(* CODESYS project Tc3_Element.library
   Description: State Model with Observer and Events
   Author: Peter Zerlauth
   Company: Zerlauth
   Version: 0.0.0.1
   Title: Tc3_Element
   DefaultNamespace: Tc3_Element
   Placeholder: Tc3_Element

Project tree, tasks and I/O mapping:
  libraries: Tc2_Standard, * (Beckhoff Automation GmbH); Tc2_System, * (Beckhoff Automation GmbH); Tc2_Utilities, * (Beckhoff Automation GmbH); Tc3_Module, 3.4.5.0 (Beckhoff Automation GmbH)
  Element/
    Event/
      Observable/
        function block FB_Observable [ST]: FB_exit, M_Attach, M_Clear, M_Detach, M_Find, M_Index, M_Notify, P_Length
        interface I_Observable: M_Attach, M_Detach, P_Length
        interface I_Observer: M_Notify
      data type E_Event
      data type E_EventType
      function block FB_Event [ST]: FB_init, M_Abort, M_AddBOOL, M_AddINT, M_AddREAL, M_AddSTRING, M_AddTIME, M_Arguments, M_Build, M_Debug, M_Error, M_Info, M_Log, M_Warning, P_Logger, P_Observer
      interface I_Event: M_Abort, M_AddBOOL, M_AddINT, M_AddREAL, M_AddSTRING, M_AddTIME, M_Debug, M_Error, M_Info, M_Warning, P_Logger, P_Observer
      data type ST_Event
      data type ST_EventFlags
    Reflection/
      function block FB_Reflection [ST]: M_GetInstance, P_Class, P_Comment, P_ID, P_Instance, P_Timestamp
      interface I_Reflection : P_Class, P_Comment, P_ID, P_Instance, P_Timestamp
    Sequence/
      data type E_Sequence
      function block FB_Sequence [ST]: FB_init, M_Await, M_Reset, M_Restore, M_Set, P_Number, P_Timeout
      interface I_Sequence: M_Await, M_Reset, M_Set, P_Number, P_Timeout
      data type ST_Sequence
      data type ST_SequenceOptions
    data type E_Request
    data type E_State
    function block FB_Element [ST]: M_Aborted, M_Aborting, M_Completed, M_Completing, M_Execute, M_Held, M_Holding, M_Idle, M_Paused, M_Pausing, M_Resetting, M_Resuming, M_Starting, M_Stopped, M_Stopping, M_Unholding, M_OnState, M_Request, P_Event, P_Reflection, P_Sequence, P_State
    interface I_Element: M_Request, P_Event, P_Reflection, P_State
  Level/
    function block FB_Level [ST]: M_Aborting, M_Attach, M_Completing, M_Detach, M_Holding, M_Pausing, M_Resetting, M_Resuming, M_Starting, M_Stopping, M_Unholding, P_List
  List/
    function block FB_ListElement [ST]: FB_exit, M_Add, M_Clear, M_Find, M_Index, M_Remove, P_Length
    function block FB_ListObject [ST]: FB_exit, M_Add, M_Clear, M_Find, M_Index, M_Remove, P_Length
    function block FB_ListString [ST]: FB_exit, M_Add, M_Clear, M_Find, M_Index, M_Remove, P_Length
    interface I_ListBase: M_Clear, P_Length
    interface I_ListElement: M_Add, M_Find, M_Index, M_Remove
    interface I_ListObject: M_Add, M_Find, M_Index, M_Remove
    interface I_ListString: M_Add, M_Find, M_Index, M_Remove
  Logger/
    function block FB_FileLogger [ST]: M_Delete, M_Find, M_Log, M_Reset
    function block FB_Logger [ST]: M_Delete, M_Find, M_Log, M_Reset
    function block FB_LoggingProvider [ST]: FB_exit, M_Add, M_Clear, M_Find, M_Index, M_Log, M_Remove, M_Reset, P_Length
    interface I_Logger: M_Log, M_Reset
  Module/
    data type E_Mode
    function block FB_Module [ST]: M_Aborting, M_Completing, M_Holding, M_Idle, M_Mode, M_OnMode, M_Resetting, M_Starting, M_Stopping, M_Unholding, P_Mode
    interface I_Module: M_Mode, P_Mode
  Object/
    function block FB_Object [ST]
    interface I_Object
  Utils/
    File/
      function block FB_File [ST]: M_Append, M_AppendLine, M_Close, M_Create, M_Delete, M_Load, M_Open, M_Read, M_Write, P_Error, P_Open
      interface I_File: M_Append, M_AppendLine, M_Close, M_Create, M_Delete, M_Load, M_Open, M_Read, M_Write, P_Error, P_Open
    function block FB_Debounce [ST]: P_Value
  Version/
    global variables Global_Version
*)

// Element/Event/E_Event
{attribute 'qualified_only'}
{attribute 'strict'}
{attribute 'to_string'}
TYPE E_Event :
(
	Verbose			:= 0,
	Debug			:= 1,
	Information		:= 2,
	Warning			:= 3,
	Error			:= 4
);
END_TYPE

// Element/Event/E_EventType
{attribute 'qualified_only'}
{attribute 'strict'}
{attribute 'to_string'}
TYPE E_EventType :
(
	Information		:= 1,
	Warning			:= 2,
	Stop			:= 3,
	Abort			:= 4
);
END_TYPE

// Element/Event/ST_Event
{attribute 'analysis' := '-33'}
TYPE ST_Event :
	STRUCT
		iSource:		I_Element;
		eEventType:		E_Event;
		tTimestamp:   	DT;
		nID:			ULINT;
		sInstance:		STRING(255);
		sClass:			STRING(255);
		sMessage:		STRING(255);
		sDefault:		STRING(255);
		sArguments:		STRING(255);
   		{attribute 'hide'} 
		stFlags:		ST_EventFlags;
	END_STRUCT
END_TYPE

// Element/Event/ST_EventFlags
{attribute 'analysis' := '-33'}
TYPE ST_EventFlags :
STRUCT
	bActive:		BIT;
	bRemove:		BIT;
END_STRUCT
END_TYPE

// Element/Sequence/E_Sequence
{attribute 'qualified_only'}
{attribute 'strict'}
{attribute 'to_string'}

TYPE E_Sequence :
(
	Undefined		:= -32767,
	Start			:= 0,
	Done			:= 32767
)INT;
END_TYPE

// Element/Sequence/ST_Sequence
TYPE ST_Sequence :
STRUCT
	sMessage:				STRING(255);
	nNumber:				INT;
END_STRUCT
END_TYPE

// Element/Sequence/ST_SequenceOptions
TYPE ST_SequenceOptions :
STRUCT
	bSaveOnStopping:		BOOL;
END_STRUCT
END_TYPE

// Element/E_Request
{attribute 'qualified_only'}
{attribute 'strict'}
{attribute 'to_string'}

TYPE E_Request :
(
	{attribute 'hide'}
    Undefined   := 0,
	{attribute 'analysis' := '-27'}
	Reset       := 1,
	{attribute 'analysis' := '-27'}
    Start       := 2,
	{attribute 'analysis' := '-27'}
	Pause		:= 4,
	{attribute 'analysis' := '-27'}
	Hold		:= 5,
	{attribute 'analysis' := '-27'}
	Complete	:= 6,
	{attribute 'analysis' := '-27'}
	Stop		:= 7,
	{attribute 'analysis' := '-27'}
	Abort		:= 8
);
END_TYPE

// Element/E_State
{attribute 'qualified_only'}
{attribute 'strict'}
{attribute 'to_string'}
TYPE E_State :
(
    Resetting       := -1,
   	Idle            := 0,
    Starting        := 1,
    Execute         := 2,
	Pausing			:= 3,
	Paused			:= 4,
	Resuming		:= 5,
	Holding			:= 6,
	Held			:= 7,
	Unholding		:= 8,
    Completing      := 9,
    Completed       := 10,
    Stopping        := 11,
    Stopped         := 12,
    Aborting        := 13,
    Aborted         := 14

)INT;
END_TYPE

// Module/E_Mode
{attribute 'qualified_only'}
{attribute 'strict'}
{attribute 'to_string'}
TYPE E_Mode :
(
	{attribute 'hide'}
    Undefined   := 0,
	Automatic   := 1,
    Semiauto    := 2,
	Manual		:= 3
);
END_TYPE

// Version/Global_Version
{attribute 'TcGenerated'}
{attribute 'no-analysis'}
{attribute 'linkalways'}
// This function has been automatically generated from the project information.
VAR_GLOBAL CONSTANT
	{attribute 'const_non_replaced'}
	stLibVersion_Tc3_Element : ST_LibVersion := (iMajor := 0, iMinor := 0, iBuild := 0, iRevision := 1, nFlags := 0, sVersion := '0.0.0.1');
END_VAR

// Element/Event/Observable/FB_Observable
FUNCTION_BLOCK PUBLIC FB_Observable IMPLEMENTS I_Observable
VAR_INPUT
	iParent:		I_Element;	
END_VAR
VAR
	bObserver:		BOOL;
	pList: 			POINTER TO I_Element;
    {attribute 'hide'}
	nLength:		DINT;
	{IF (defined (release))}
    	{attribute 'hide'}
	{END_IF}
	aList:			POINTER TO POINTER TO ARRAY [0..100] OF I_Element:=ADR(pList);
END_VAR

// https://peterzerlauth.com/
bObserver:= TRUE;

METHOD FB_exit : BOOL
VAR_INPUT
	bInCopyCode : BOOL; // if TRUE, the exit method is called for exiting an instance that is copied afterwards (online change).
END_VAR
M_Clear();
END_METHOD

METHOD M_Attach : BOOL
VAR_INPUT
	iObject: 	I_Element;
END_VAR
VAR
	pOldList: 	POINTER TO I_Element;
END_VAR
IF iObject <> 0 THEN
	// First Item
	IF pList = 0 THEN
		nLength:= nLength + 1;
		pList:= __NEW(POINTER TO I_Element,DINT_TO_UDINT(nLength));
	ELSE
		// Item already in List
		IF M_Find(iObject) = -1 THEN
			// backup 
			pOldList:= pList;
			// new Length
			nLength:= nLength + 1;
			// new pointer
			pList:= __NEW(POINTER TO I_Element,DINT_TO_UDINT(nLength));
			// restore
			Memcpy(pList,pOldList, SIZEOF(POINTER TO I_Element)*DINT_TO_UDINT(nLength -1));
			// delete old
			__DELETE(pOldList);
		ELSE
			M_Attach:= FALSE;	
			RETURN;
		END_IF
	END_IF
	IF pList = 0 THEN
		RETURN;
	END_IF
	// add new Object
	pList[nLength-1]:= iObject;
	M_Attach:= TRUE;
ELSE
	M_Attach:= FALSE;	
END_IF
END_METHOD

METHOD M_Clear
IF pList <> 0 THEN
	nLength:= 0;
	__DELETE(pList);
END_IF
END_METHOD

METHOD M_Detach : BOOL
VAR_INPUT
	iObject: 	I_Element;
END_VAR
VAR
	pOldList:			POINTER TO I_Element;
	nPosition: 			DINT;
END_VAR
IF iObject <> 0 THEN
	// First Item
	IF nLength >= 0 THEN
		// Item already in List
		nPosition:= M_Find(iObject);
		IF nPosition <> -1 THEN
			// backup 
			pOldList:= pList;
			// new Length
			nLength:= nLength -1;
			// new pointer
			pList:= __NEW(POINTER TO I_Element,DINT_TO_UDINT(nLength));
			// restore lower part
			Memcpy(pList,pOldList, SIZEOF(POINTER TO I_Element) * DINT_TO_UDINT(nPosition));
			//pList[nPosition]:= iObject;
			Memcpy(pList + (SIZEOF(POINTER TO I_Element)*nPosition),pOldList + (SIZEOF(POINTER TO I_Element)*(nPosition + 1)), SIZEOF(POINTER TO I_Element) * DINT_TO_UDINT(nLength - nPosition));
			// delete old
			__DELETE(pOldList);
		ELSE
			M_Detach:= FALSE;	
			RETURN;
		END_IF
	ELSE
		M_Detach:= FALSE;	
		RETURN;
	END_IF
	M_Detach:= TRUE;
ELSE
	M_Detach:= FALSE;	
END_IF
END_METHOD

METHOD M_Find : DINT
VAR_INPUT
	iObject: 	I_Element;
END_VAR
VAR
	nIndex: 	UINT;
END_VAR
// Object already in List
M_Find := -1;
WHILE nIndex < nLength DO
    IF (pList[nIndex] = iObject) THEN
        M_Find := nIndex;
        RETURN;
    END_IF
	nIndex := nIndex + 1;
END_WHILE
END_METHOD

METHOD M_Index : I_Observer
VAR_INPUT
	nIndex: 	DINT;
END_VAR
IF nIndex <= nLength THEN
	M_Index:= pList[nIndex].P_Event.P_Observer;
END_IF
END_METHOD

METHOD M_Notify
VAR_INPUT
	iSender:		I_Element;
END_VAR

VAR
	nIndex: 		DINT;
END_VAR
iParent.M_Request(E_Request.Abort);
IF bObserver THEN
	bObserver:= FALSE;
	WHILE nIndex < nLength DO
		pList[nIndex].P_Event.P_Observer.M_Notify(iSender);	
		nIndex:= nIndex + 1; 
	END_WHILE
	
END_IF
END_METHOD

{attribute 'OPC.UA.DA.Property' := '1'}
{attribute 'monitoring' := 'call'}
PROPERTY P_Length : DINT
GET
P_Length:= nLength;
END_GET
END_PROPERTY

END_FUNCTION_BLOCK

// Element/Event/Observable/I_Observable
INTERFACE I_Observable EXTENDS I_Observer

METHOD PUBLIC M_Attach : BOOL
VAR_INPUT
	iObject: 	I_Element;
END_VAR
END_METHOD

METHOD PUBLIC M_Detach : BOOL
VAR_INPUT
	iObject: 	I_Element;
END_VAR
END_METHOD

{attribute 'OPC.UA.DA.Property' := '1'}
{attribute 'monitoring' := 'call'}
PROPERTY P_Length : DINT
GET
END_GET
END_PROPERTY

END_INTERFACE

// Element/Event/Observable/I_Observer
INTERFACE I_Observer EXTENDS I_Object

METHOD PUBLIC M_Notify
VAR_INPUT
	iSender:		I_Element;
END_VAR
END_METHOD

END_INTERFACE

// Object/I_Object
INTERFACE I_Object EXTENDS __SYSTEM.IQueryInterface

END_INTERFACE

// Element/I_Element
INTERFACE I_Element EXTENDS I_Object

METHOD PUBLIC M_Request : BOOL
VAR_INPUT
	eRequest:	E_Request;
END_VAR
END_METHOD

PROPERTY PUBLIC P_Event : I_Event
GET
END_GET
END_PROPERTY

PROPERTY PUBLIC P_Reflection : I_Reflection
GET
END_GET
END_PROPERTY

PROPERTY PUBLIC P_State : E_State
GET
END_GET
END_PROPERTY

END_INTERFACE

// Element/Event/I_Event
INTERFACE I_Event EXTENDS I_Object

METHOD PUBLIC M_Abort
VAR_INPUT
	sMessage:				STRING(255);
	nID:					ULINT;
END_VAR
END_METHOD

METHOD PUBLIC M_AddBOOL : I_Event
VAR_INPUT
	Value: 	BOOL;
END_VAR
END_METHOD

METHOD PUBLIC M_AddINT : I_Event
VAR_INPUT
	Value: 	LINT;
END_VAR
END_METHOD

METHOD PUBLIC M_AddREAL : I_Event
VAR_INPUT
	Value: 	Lreal;
	Decimals: INT;
END_VAR
END_METHOD

METHOD PUBLIC M_AddSTRING : I_Event
VAR_INPUT
	Value: STRING(255);
END_VAR
END_METHOD

METHOD PUBLIC M_AddTIME : I_Event
VAR_INPUT
	Value: 	TIME;
END_VAR
END_METHOD

METHOD PUBLIC M_Debug
VAR_INPUT
	sMessage:				STRING(255);
END_VAR
END_METHOD

METHOD PUBLIC M_Error
VAR_INPUT
	sMessage:				STRING(255);
	nID:					ULINT;
END_VAR
END_METHOD

METHOD PUBLIC M_Info
VAR_INPUT
	sMessage:				STRING(255);
	nID:					ULINT;
END_VAR
END_METHOD

METHOD PUBLIC M_Warning
VAR_INPUT
	sMessage:				STRING(255);
	nID:					ULINT;
END_VAR
END_METHOD

{attribute 'OPC.UA.DA.Property' := '1'}
{attribute 'monitoring' := 'call'}
PROPERTY PUBLIC P_Logger : I_Logger
GET
END_GET
SET
END_SET
END_PROPERTY

{attribute 'OPC.UA.DA.Property' := '1'}
{attribute 'monitoring' := 'call'}
PROPERTY PUBLIC P_Observer : I_Observable
GET
END_GET
END_PROPERTY

END_INTERFACE

// Logger/I_Logger
INTERFACE I_Logger EXTENDS I_Object

METHOD PUBLIC M_Log
VAR_INPUT
	{attribute 'analysis' := '-33'}
	stEvent	: ST_Event;
END_VAR
END_METHOD

METHOD PUBLIC M_Reset
VAR_INPUT
END_VAR
END_METHOD

END_INTERFACE

// Element/Event/FB_Event
FUNCTION_BLOCK FB_Event IMPLEMENTS I_Event
VAR_INPUT
	fbObserver:			FB_Observable;				// Observer
END_VAR
VAR_OUTPUT
END_VAR
VAR
	{IF (defined (release))}
    	{attribute 'hide'}
	{END_IF}
	iLogger:			I_Logger;					// Event logger
	{IF (defined (release))}
    	{attribute 'hide'}
	{END_IF}
	iParent:			I_Element;					// Parent component
	{IF (defined (release))}
    	{attribute 'hide'}
	{END_IF}
	fbList:				FB_ListString;				// contains a list with string values
	stDebug:			ST_Event;					// last debug event
	stInfo:				ST_Event;					// last info event
	stWarning:			ST_Event;					// last warning event
	stError:			ST_Event;					// last stop event
	stAbort:			ST_Event;					// last abort event
END_VAR

// https://peterzerlauth.com/
fbObserver();

METHOD FB_init : BOOL
VAR_INPUT
	bInitRetains : BOOL; // if TRUE, the retain variables are initialized (warm start / cold start)
	bInCopyCode : BOOL;  // if TRUE, the instance afterwards gets moved into the copy code (online change)
	iParent:			I_Element;
END_VAR
THIS^.iParent:= iParent;
fbObserver.iParent:= iParent;
END_METHOD

METHOD PUBLIC M_Abort
VAR_INPUT
	sMessage:				STRING(255);
	nID:					ULINT;
END_VAR
stAbort.sMessage:= sMessage;
stAbort.iSource:= iParent;
stAbort.sInstance:= iParent.P_Reflection.P_Instance;
stAbort.sClass:= iParent.P_Reflection.P_Class;
stAbort.eEventType:= E_Event.Error;
stAbort.tTimestamp:= iParent.P_Reflection.P_Timestamp;
stAbort.nID:= nID;
stAbort.sDefault:= M_Build(sMessage);
stAbort.sArguments:= M_Arguments();
stAbort.stFlags.bActive:= TRUE;
stAbort.stFlags.bRemove:= FALSE;

IF iLogger = 0 THEN
	M_Log(stAbort);
ELSE
	iLogger.M_Log(stAbort);
END_IF

fbObserver.M_Notify(iParent);
END_METHOD

METHOD PUBLIC M_AddBOOL : I_Event
VAR_INPUT
	Value: 	bool;
END_VAR
fbList.M_Add(BOOL_TO_STRING(Value));
M_AddBOOL:= THIS^;
END_METHOD

METHOD PUBLIC M_AddINT : I_Event
VAR_INPUT
	Value: 	LINT;
END_VAR
fbList.M_Add(LINT_TO_STRING(Value));
M_AddINT:= THIS^;
END_METHOD

METHOD PUBLIC M_AddREAL : I_Event
VAR_INPUT
	Value: 	Lreal;
	Decimals: INT;
END_VAR
fbList.M_Add(LREAL_TO_FMTSTR(Value, Decimals, TRUE));
M_AddREAL:= THIS^;
END_METHOD

METHOD PUBLIC M_AddSTRING : I_Event
VAR_INPUT
	Value: STRING(255);
END_VAR
fbList.M_Add(Value);
M_AddSTRING:= THIS^;
END_METHOD

METHOD PUBLIC M_AddTIME : I_Event
VAR_INPUT
	Value: 	TIME;
END_VAR
fbList.M_Add(TIME_TO_STRING(Value));
M_AddTIME:= THIS^;
END_METHOD

METHOD INTERNAL M_Arguments : STRING(255)
VAR_INPUT
END_VAR
VAR
	nIndex:			INT;
END_VAR
WHILE nIndex < fbList. P_Length DO
	M_Arguments:= Concat(Concat(M_Arguments, fbList.M_Index(nIndex)), '$N');
	nIndex:= nIndex + 1;
END_WHILE

fbList.M_Clear();
END_METHOD

METHOD INTERNAL M_Build : STRING(255)
VAR_INPUT
	sMessage:		STRING(255);
END_VAR
VAR
	nIndex:		   	DINT;
	nPosition: 		INT;
END_VAR
nPosition:= Find(sMessage, '%s');
WHILE nPosition <> 0 DO
	sMessage:= Replace(sMessage, fbList.M_Index(nIndex), 2, nPosition);
	nPosition:= Find(sMessage, '%s');
	nIndex:= nIndex + 1;
END_WHILE
M_Build:= sMessage;
END_METHOD

METHOD PUBLIC M_Debug
VAR_INPUT
	sMessage:				STRING(255);
END_VAR
stDebug.sMessage:= sMessage;
stDebug.iSource:= iParent;
stDebug.sInstance:= iParent.P_Reflection.P_Instance;
stDebug.sClass:= iParent.P_Reflection.P_Class;
stDebug.eEventType:= E_Event.Debug;
stDebug.tTimestamp:= iParent.P_Reflection.P_Timestamp;
stDebug.nID:= 0;
stDebug.sDefault:= M_Build(sMessage);
stDebug.sArguments:= M_Arguments();
stDebug.stFlags.bActive:= TRUE;
stDebug.stFlags.bRemove:= TRUE;

IF iLogger = 0 THEN
	M_Log(stDebug);
ELSE
	iLogger.M_Log(stDebug);
END_IF
END_METHOD

METHOD PUBLIC M_Error
VAR_INPUT
	sMessage:				STRING(255);
	nID:					ULINT;
END_VAR
stError.sMessage:= sMessage;
stError.iSource:= iParent;
stError.sInstance:= iParent.P_Reflection.P_Instance;
stError.sClass:= iParent.P_Reflection.P_Class;
stError.eEventType:= E_Event.Error;
stError.tTimestamp:= iParent.P_Reflection.P_Timestamp;
stError.nID:= nID;
stError.sDefault:= M_Build(sMessage);
stError.sArguments:= M_Arguments();
stError.stFlags.bActive:= TRUE;
stError.stFlags.bRemove:= FALSE;

IF iLogger = 0 THEN
	M_Log(stError);
ELSE
	iLogger.M_Log(stError);
END_IF
END_METHOD

METHOD PUBLIC M_Info
VAR_INPUT
	sMessage:				STRING(255);
	nID:					ULINT;
END_VAR
stInfo.sMessage:= sMessage;
stInfo.iSource:= iParent;
stInfo.sInstance:= iParent.P_Reflection.P_Instance;
stInfo.sClass:= iParent.P_Reflection.P_Class;
stInfo.eEventType:= E_Event.Information;
stInfo.tTimestamp:= iParent.P_Reflection.P_Timestamp;
stInfo.nID:= nID;
stInfo.sDefault:= M_Build(sMessage);
stInfo.sArguments:= M_Arguments();
stInfo.stFlags.bActive:= TRUE;
stInfo.stFlags.bRemove:= TRUE;

IF iLogger = 0 THEN
	M_Log(stInfo);
ELSE
	iLogger.M_Log(stInfo);
END_IF
END_METHOD

METHOD PRIVATE M_Log : BOOL
VAR_INPUT
	stEvent	: ST_Event;
END_VAR
END_METHOD

METHOD PUBLIC M_Warning
VAR_INPUT
	sMessage:				STRING(255);
	nID:					ULINT;
END_VAR
stWarning.sMessage:= sMessage;
stWarning.iSource:= iParent;
stWarning.sInstance:= iParent.P_Reflection.P_Instance;
stWarning.sClass:= iParent.P_Reflection.P_Class;
stWarning.eEventType:= E_Event.Warning;
stWarning.tTimestamp:= iParent.P_Reflection.P_Timestamp;
stWarning.nID:= nID;
stWarning.sDefault:= M_Build(sMessage);
stWarning.sArguments:= M_Arguments();
stWarning.stFlags.bActive:= TRUE;
stWarning.stFlags.bRemove:= TRUE;

IF iLogger = 0 THEN
	M_Log(stWarning);
ELSE
	iLogger.M_Log(stWarning);
END_IF
END_METHOD

{attribute 'OPC.UA.DA.Property' := '1'}
{attribute 'monitoring' := 'call'}
PROPERTY P_Logger : I_Logger
GET
P_Logger:= iLogger;
END_GET
SET
iLogger:= P_Logger;
END_SET
END_PROPERTY

{attribute 'OPC.UA.DA.Property' := '1'}
{attribute 'monitoring' := 'call'}
PROPERTY PUBLIC P_Observer : I_Observable
GET
P_Observer:= fbObserver;
END_GET
END_PROPERTY

END_FUNCTION_BLOCK

// List/FB_ListString
{attribute 'no_explicit_call' := 'do not call this POU directly'} 
FUNCTION_BLOCK FB_ListString IMPLEMENTS I_ListString
VAR
	pList: 			POINTER TO STRING(255);
	{IF (defined (release))}
    	{attribute 'hide'}
	{END_IF}
	aList:			POINTER TO POINTER TO ARRAY [0..24] OF STRING(255):=ADR(pList);
END_VAR
VAR_OUTPUT
	{IF (defined (release))}
    	{attribute 'hide'}
	{END_IF}
	nLength:		INT;	
END_VAR

// https://peterzerlauth.com/

METHOD FB_exit : BOOL
VAR_INPUT
	bInCopyCode : BOOL; // if TRUE, the exit method is called for exiting an instance that is copied afterwards (online change).
END_VAR
M_Clear();
END_METHOD

METHOD PUBLIC M_Add : BOOL
VAR_INPUT
	Object: 	STRING(255);
END_VAR
VAR
	pOldList: 	POINTER TO STRING(255);
END_VAR
IF LEN(Object) <> 0 THEN
	// First Item
	IF pList = 0 THEN
		nLength:= nLength + 1;
		pList:= __NEW(STRING(255),DINT_TO_UDINT(nLength));
	ELSE
		// Item already in List
		IF M_Find(Object) = -1 THEN
			// backup 
			pOldList:= pList;
			// new Length
			nLength:= nLength + 1;
			// new pointer
			pList:= __NEW(STRING(255),DINT_TO_UDINT(nLength));
			// restore
			Memcpy(pList,pOldList, SIZEOF(STRING(255))*DINT_TO_UDINT(nLength -1));
			// delete old
			__DELETE(pOldList);
		ELSE
			M_Add:= FALSE;	
			RETURN;
		END_IF
	END_IF
	IF pList = 0 THEN
		RETURN;
	END_IF
	// add new Object
	pList[nLength-1]:= Object;
	M_Add:= TRUE;
ELSE
	M_Add:= FALSE;	
END_IF
END_METHOD

METHOD PUBLIC M_Clear : BOOL
IF pList <> 0 THEN
	nLength:= 0;
	__DELETE(pList);
END_IF
M_Clear:= TRUE;
END_METHOD

METHOD PUBLIC M_Find : DINT
VAR_INPUT
	Object: 	STRING(255);
END_VAR
VAR
	nIndex: 	UINT;
END_VAR
// Object already in List
M_Find := -1;
WHILE nIndex < nLength DO
    IF (pList[nIndex] = Object) THEN
        M_Find := nIndex;
        RETURN;
    END_IF
	nIndex := nIndex + 1;
END_WHILE
END_METHOD

METHOD PUBLIC M_Index : STRING(255)
VAR_INPUT
	Index: 	DINT;
END_VAR
IF pList <> 0 THEN
	IF Index <= nLength THEN
		M_Index:= pList[Index];
	ELSE
		M_Index:= '';
	END_IF
ELSE
	M_Index:= '';
END_IF
END_METHOD

METHOD PUBLIC M_Remove : BOOL
VAR_INPUT
	Object: 	STRING(255);
END_VAR
VAR
	pOldList:			POINTER TO STRING(255);
	nPosition: 			DINT;
END_VAR
IF Object <> '' THEN
	// First Item
	IF nLength >= 0 THEN
		// Item already in List
		nPosition:= M_Find(Object);
		IF nPosition <> -1 THEN
			// backup 
			pOldList:= pList;
			// new Length
			nLength:= nLength -1;
			// new pointer
			pList:= __NEW(POINTER TO I_Object,DINT_TO_UDINT(nLength));
			// restore lower part
			Memcpy(pList,pOldList, SIZEOF(STRING(255)) * DINT_TO_UDINT(nPosition));
			//pList[nPosition]:= iObject;
			Memcpy(pList + (SIZEOF(STRING(255))*nPosition),pOldList + (SIZEOF(STRING(255))*(nPosition + 1)), SIZEOF(STRING(255)) * DINT_TO_UDINT(nLength - nPosition));
			// delete old
			__DELETE(pOldList);
		ELSE
			M_Remove:= FALSE;	
			RETURN;
		END_IF
	ELSE
		M_Remove:= FALSE;	
		RETURN;
	END_IF
	M_Remove:= TRUE;
ELSE
	M_Remove:= FALSE;	
END_IF
END_METHOD

{attribute 'OPC.UA.DA.Property' := '1'}
{attribute 'monitoring' := 'call'}
PROPERTY PUBLIC P_Length : DINT
GET
P_Length:= nLength;
END_GET
END_PROPERTY

END_FUNCTION_BLOCK

// List/I_ListString
INTERFACE I_ListString EXTENDS I_ListBase

METHOD PUBLIC M_Add : BOOL
VAR_INPUT
	Object: 	STRING(255);
END_VAR
END_METHOD

METHOD PUBLIC M_Find : DINT
VAR_INPUT
	Object: 	STRING(255);
END_VAR
END_METHOD

METHOD PUBLIC M_Index : STRING(255)
VAR_INPUT
	Index: 	DINT;
END_VAR
END_METHOD

METHOD PUBLIC M_Remove : BOOL
VAR_INPUT
	Object: 	STRING(255);
END_VAR
END_METHOD

END_INTERFACE

// List/I_ListBase
INTERFACE I_ListBase EXTENDS I_Object

METHOD PUBLIC M_Clear : BOOL
END_METHOD

{attribute 'OPC.UA.DA.Property' := '1'}
{attribute 'monitoring' := 'call'}
PROPERTY public P_Length : DINT
GET
END_GET
END_PROPERTY

END_INTERFACE

// Element/Reflection/FB_Reflection
{attribute 'reflection'} 
FUNCTION_BLOCK PUBLIC FB_Reflection IMPLEMENTS I_Reflection
VAR_INPUT
END_VAR
VAR_OUTPUT
END_VAR
VAR
	sIdentifier:						STRING(25):= 'Undefined';		// Identifier
	{attribute 'instance-path'}                                     	
    {attribute 'noinit'}                                            	
    sInstancePath:						STRING(255);					// Instance-Path
	fbReadSymInfo: 						PLC_ReadSymInfoByNameEx;		// Read symbol infos
END_VAR                                                             	
VAR_STAT                                                            	
	nCycle: 							UDINT;							// Cycle counter
	fbGetTime:							NT_GetTime;
END_VAR

// https://peterzerlauth.com/

// Update once for all function blocks
IF nCycle <> TwinCAT_SystemInfoVarList._TaskInfo[GETCURTASKINDEXEX()].CycleCount THEN
	nCycle:= TwinCAT_SystemInfoVarList._TaskInfo[GETCURTASKINDEXEX()].CycleCount;
	fbGetTime(Start:= TRUE);
END_IF

// Read symbol information
IF NOT fbReadSymInfo.START THEN
	M_GetInstance();
	fbReadSymInfo.PORT:= TwinCAT_SystemInfoVarList._AppInfo.AdsPort;
	fbReadSymInfo.START:= TRUE;
END_IF
fbReadSymInfo();

METHOD PROTECTED M_GetInstance
VAR_INPUT
END_VAR
VAR
    sName:				STRING(255);
    nPosition:			INT;
END_VAR
sName := CONCAT(TwinCAT_SystemInfoVarList._AppInfo.ProjectName, '.');

nPosition := FIND(sInstancePath, sName);
IF nPosition > 0 THEN
    fbReadSymInfo.SYMNAME:= DELETE(sInstancePath, nPosition-1 + LEN(sName), 1);
END_IF

nPosition := FIND(fbReadSymInfo.SYMNAME, sName);

IF nPosition > 0 THEN
    fbReadSymInfo.SYMNAME:= DELETE(fbReadSymInfo.SYMNAME, nPosition - 1 + LEN(sName), 1);
END_IF

fbReadSymInfo.SYMNAME:= Left(fbReadSymInfo.SYMNAME, LEN(fbReadSymInfo.SYMNAME) - LEN('.fbReflection'));
END_METHOD

{attribute 'OPC.UA.DA.Property' := '1'}
{attribute 'monitoring' := 'call'}
PROPERTY PUBLIC P_Class : STRING(255)
GET
{attribute 'OPC.UA.DA.Property' := '1'}
{attribute 'monitoring' := 'call'}
VAR
END_VAR
P_Class:= fbReadSymInfo.SYMINFO.symDataType;
END_GET
END_PROPERTY

{attribute 'OPC.UA.DA.Property' := '1'}
{attribute 'monitoring' := 'call'}
PROPERTY PUBLIC P_Comment : STRING(255)
GET
P_Comment:= fbReadSymInfo.SYMINFO.symComment;
END_GET
END_PROPERTY

{attribute 'OPC.UA.DA.Property' := '1'}
{attribute 'monitoring' := 'call'}
PROPERTY PUBLIC P_ID : STRING(25)
GET
P_ID:= sIdentifier;
END_GET
SET
PUBLIC 
VAR
END_VAR
sIdentifier:= P_ID;
END_SET
END_PROPERTY

{attribute 'OPC.UA.DA.Property' := '1'}
{attribute 'monitoring' := 'call'}
PROPERTY PUBLIC P_Instance : STRING(255)
GET
P_Instance:= fbReadSymInfo.SYMNAME;
END_GET
END_PROPERTY

{attribute 'OPC.UA.DA.Property' := '1'}
{attribute 'monitoring' := 'call'}
PROPERTY PUBLIC P_Timestamp : DT
GET
P_Timestamp:= SYSTEMTIME_TO_DT(fbGetTime.TIMESTR);
END_GET
END_PROPERTY

END_FUNCTION_BLOCK

// Element/Reflection/I_Reflection 
INTERFACE I_Reflection EXTENDS I_Object

{attribute 'OPC.UA.DA.Property' := '1'}
{attribute 'monitoring' := 'call'}
PROPERTY PUBLIC P_Class : STRING(255)
GET
END_GET
END_PROPERTY

{attribute 'OPC.UA.DA.Property' := '1'}
{attribute 'monitoring' := 'call'}
PROPERTY PUBLIC P_Comment : STRING(255)
GET
END_GET
END_PROPERTY

{attribute 'OPC.UA.DA.Property' := '1'}
{attribute 'monitoring' := 'call'}
PROPERTY PUBLIC P_ID : STRING(25)
GET
END_GET
SET
END_SET
END_PROPERTY

{attribute 'OPC.UA.DA.Property' := '1'}
{attribute 'monitoring' := 'call'}
PROPERTY PUBLIC P_Instance : STRING(255)
GET
END_GET
END_PROPERTY

{attribute 'OPC.UA.DA.Property' := '1'}
{attribute 'monitoring' := 'call'}
PROPERTY PUBLIC P_Timestamp : DT
GET
END_GET
END_PROPERTY

END_INTERFACE

// Element/Sequence/FB_Sequence
FUNCTION_BLOCK FB_Sequence IMPLEMENTS I_Sequence
VAR_INPUT
	bHeld:				BOOL;
END_VAR
VAR_OUTPUT
	bTimeout:			BOOL;
END_VAR
VAR
	iParent:			I_Element;
	stExecute:			ST_Sequence;
	stLast:				ST_Sequence;
	stActual:			ST_Sequence;
	fbTimeout:			TON;
	fbDelay: 			TON;
END_VAR

// https://peterzerlauth.com/

METHOD FB_init : BOOL
VAR_INPUT
	bInitRetains : BOOL; // if TRUE, the retain variables are initialized (warm start / cold start)
	bInCopyCode : BOOL;  // if TRUE, the instance afterwards gets moved into the copy code (online change)
	iParent:			I_Element;
END_VAR
THIS^.iParent:= iParent;
END_METHOD

METHOD PUBLIC M_Await : BOOL
VAR_INPUT
	sMessage:				STRING(255);
	nID:					ULINT;
	tTimeout:				TIME;
	tDelay:					TIME;	
	bPause:					BOOL;
	bReturn:				BOOL;
	nNumber:				INT;
END_VAR
// Assign the current message to the actual status structure
stActual.sMessage := sMessage;  

// Check the return condition
IF bReturn THEN  
    // Reset timeout
    fbTimeout(IN := FALSE);  
    bTimeout := FALSE; 
    // Start delay
    fbDelay(IN := TRUE, PT := tDelay);  
    
    // Delay elapsed  
    IF fbDelay.Q THEN  
        M_Await := TRUE;  
        // Set the next step number
        stActual.nNumber := nNumber;   
        // Save the last known state  
        stLast := stActual;  
        // Last state to restore
        IF iParent.P_State = E_State.Execute THEN  
            stExecute := stLast;  
        END_IF  
        
        // Reset delay
        fbDelay(IN := FALSE);  
//         IF bHeld THEN  
//             // Request a hold operation to the parent  
//             iParent.M_Request(E_Request.Hold);  
//         ELSIF bPause THEN  
//             // Request a pause operation to the parent  
//             iParent.M_Request(E_Request.Pause);  
//         END_IF  
    END_IF  

ELSE  
    // Reset delay
    fbDelay(IN := FALSE);  
    // Start timeout
    fbTimeout(IN := tTimeout <> T#0S, PT := tTimeout);  
    // Timeout elapsed
    IF fbTimeout.Q THEN
		bTimeout := TRUE;   
        // Report Timeout 
        iParent.P_Event.M_Error(sMessage, nID);  
    END_IF  
END_IF
END_METHOD

METHOD PUBLIC M_Reset : BOOL
VAR_INPUT
END_VAR
bTimeout:= FALSE;
fbDelay(IN:= FALSE);
fbTimeout(IN:= FALSE);
stActual.sMessage:= 'fbSequence.M_Reset()';
stActual.nNumber:= E_Sequence.Start;
M_Reset:= TRUE;
END_METHOD

METHOD PUBLIC M_Restore : BOOL
VAR_INPUT
END_VAR
stLast:= stActual;
stActual:= stExecute;
END_METHOD

METHOD PUBLIC M_Set : BOOL
VAR_INPUT
	sMessage:				STRING(255);	
	nNumber:				INT;
END_VAR
stLast:= stActual;
IF iParent.P_State = E_State.Execute THEN
	stExecute:= stActual;
END_IF
stActual.sMessage:= Concat('Sequence.M_Set: ', sMessage);
stActual.nNumber:= nNumber;
M_Set:= TRUE;
END_METHOD


PROPERTY PUBLIC P_Number : INT
GET
P_Number:= stActual.nNumber;
END_GET
END_PROPERTY

PROPERTY PUBLIC P_Timeout : Bool
GET
P_Timeout:= bTimeout;
END_GET
END_PROPERTY

END_FUNCTION_BLOCK

// Element/Sequence/I_Sequence
INTERFACE I_Sequence EXTENDS I_Object

METHOD PUBLIC M_Await : BOOL
VAR_INPUT
	sMessage:				STRING(255);
	nID:					ULINT;
	tTimeout:				TIME;
	tDelay:					TIME;	
	bPause:					BOOL;
	bReturn:				BOOL;
	nNumber:				INT;
END_VAR
END_METHOD

METHOD PUBLIC M_Reset : BOOL
VAR_INPUT
END_VAR
END_METHOD

METHOD PUBLIC M_Set : BOOL
VAR_INPUT
	sMessage:				STRING(255);	
	nNumber:				INT;
END_VAR
END_METHOD


PROPERTY PUBLIC P_Number : INT
GET
END_GET
END_PROPERTY

PROPERTY PUBLIC P_Timeout : Bool
GET
END_GET
END_PROPERTY

END_INTERFACE

// Element/FB_Element
FUNCTION_BLOCK FB_Element IMPLEMENTS I_Element
VAR_INPUT
END_VAR
VAR_OUTPUT
END_VAR
VAR
	fbReflection:					FB_Reflection;					// Info about function block
	fbEvent:						FB_Event(THIS^);			// Event Publisher
	fbSequence:						FB_Sequence(THIS^);			// Sequence
	{attribute 'OPC.UA.DA' := '1'}
	{attribute 'OPC.UA.DA.Access' := '1'}
	eStateRequest:					E_Request;					// State command
	{attribute 'OPC.UA.DA' := '1'}
	{attribute 'OPC.UA.DA.Access' := '2'}
	eState:							E_State;					// Current state
    {attribute 'hide'}
	eStatePrevious:					E_State;					// Previous state
END_VAR

// Essential functions for event handling
fbReflection();
fbEvent();
fbSequence();

// State machine logic
CASE eState OF

    // Idle state:
    E_State.Idle:
        IF M_Idle() THEN
            eState := E_State.Starting;
        END_IF

    // Starting state:
    E_State.Starting:
        IF M_Starting() THEN
            eState := E_State.Execute;
        END_IF

    // Execute state:
    E_State.Execute:
        IF M_Execute() THEN
            eState := E_State.Completing;
        END_IF

    // Pausing state:
    E_State.Pausing:
        IF M_Pausing() THEN
            eState := E_State.Paused;
        END_IF

    // Paused state:
    E_State.Paused:
        IF M_Paused() THEN
            eState := E_State.Resuming;
        END_IF

    // Resuming state:
    E_State.Resuming:
        IF M_Resuming() THEN
            eState := E_State.Execute;
        END_IF

    // Holding state:
    E_State.Holding:
        IF M_Holding() THEN
            eState := E_State.Held;
        END_IF

    // Held state:
    E_State.Held:
        IF M_Held() THEN
            eState := E_State.Unholding;
        END_IF

    // Unholding state:
    E_State.Unholding:
        IF M_Held() THEN
            eState := E_State.Execute;
        END_IF

    // Completing state:
    E_State.Completing:
        IF M_Completing() THEN
            eState := E_State.Completed;
        END_IF

    // Completed state:
    E_State.Completed:
        IF M_Completed() THEN
            eState := E_State.Resetting;
        END_IF

    // Stopping state:
    E_State.Stopping:
        IF M_Stopping() THEN
            eState := E_State.Stopped;
        END_IF

    // Stopped state:
    E_State.Stopped:
        IF M_Stopped() THEN
            eState := E_State.Resetting;
        END_IF

    // Aborting state:
    E_State.Aborting:
        IF M_Aborting() THEN
            eState := E_State.Aborted;
        END_IF

    // Aborted state:
    E_State.Aborted:
        IF M_Aborted() THEN
            eState := E_State.Resetting;
        END_IF

    // Resetting state:
    E_State.Resetting:
        IF M_Resetting() THEN
            eState := E_State.Idle;
        END_IF

END_CASE

// handle state requests
CASE eState OF

    // Idle state:
    E_State.Idle:
        CASE eStateRequest OF
            E_Request.Start:
                eState := E_State.Starting;
            E_Request.Stop:
                eState := E_State.Stopping;
            E_Request.Abort:
                eState := E_State.Aborting;
        END_CASE

    // Starting state:
    E_State.Starting:
        CASE eStateRequest OF
            E_Request.Stop:
                eState := E_State.Stopping;
            E_Request.Abort:
                eState := E_State.Aborting;
        END_CASE

    // Execute state:
    E_State.Execute:
        CASE eStateRequest OF
            E_Request.Pause:
                eState := E_State.Pausing;
            E_Request.Hold:
                eState := E_State.Holding;
            E_Request.Stop:
                eState := E_State.Stopping;
            E_Request.Abort:
                eState := E_State.Aborting;
        END_CASE

    // Pausing state:
    E_State.Pausing:
        CASE eStateRequest OF
            E_Request.Hold:
                eState := E_State.Holding;
            E_Request.Stop:
                eState := E_State.Stopping;
            E_Request.Abort:
                eState := E_State.Aborting;
        END_CASE

    // Paused state:
    E_State.Paused:
        CASE eStateRequest OF
            E_Request.Start:
                eState := E_State.Resuming;
            E_Request.Hold:
                eState := E_State.Holding;
            E_Request.Stop:
                eState := E_State.Stopping;
            E_Request.Abort:
                eState := E_State.Aborting;
        END_CASE

    // Resuming state:
    E_State.Resuming:
        CASE eStateRequest OF
            E_Request.Hold:
                eState := E_State.Holding;
            E_Request.Stop:
                eState := E_State.Stopping;
            E_Request.Abort:
                eState := E_State.Aborting;
        END_CASE

    // Holding state:
    E_State.Holding:
        CASE eStateRequest OF
            E_Request.Stop:
                eState := E_State.Stopping;
            E_Request.Abort:
                eState := E_State.Aborting;
        END_CASE

    // Held state:
    E_State.Held:
        CASE eStateRequest OF
            E_Request.Start:
                eState := E_State.Unholding;
            E_Request.Stop:
                eState := E_State.Stopping;
            E_Request.Abort:
                eState := E_State.Aborting;
        END_CASE

    // Unholding state:
    E_State.Unholding:
        CASE eStateRequest OF
            E_Request.Stop:
                eState := E_State.Stopping;
            E_Request.Abort:
                eState := E_State.Aborting;
        END_CASE

    // Completing state:
    E_State.Completing:
        CASE eStateRequest OF
            E_Request.Stop:
                eState := E_State.Stopping;
            E_Request.Abort:
                eState := E_State.Aborting;
        END_CASE

    // Completed state:
    E_State.Completed:

    // Stopping state:
    E_State.Stopping:
        CASE eStateRequest OF
            E_Request.Abort:
                eState := E_State.Aborting;
        END_CASE

    // Stopped state:
    E_State.Stopped:
        CASE eStateRequest OF
            E_Request.Reset:
                eState := E_State.Resetting;
            E_Request.Abort:
                eState := E_State.Aborting;
        END_CASE

    // Aborting state:
	E_State.Aborting:
	
    // Aborted state:
    E_State.Aborted:
        CASE eStateRequest OF
            E_Request.Reset:
                eState := E_State.Resetting;
        END_CASE

    // Resetting state:
    E_State.Resetting:
        CASE eStateRequest OF
            E_Request.Stop:
                eState := E_State.Stopping;
            E_Request.Abort:
                eState := E_State.Aborting;
        END_CASE

END_CASE
eStateRequest := E_Request.Undefined;

// Detect state transitions and trigger event callback
IF eStatePrevious <> eState THEN
    M_OnState(eState, eStatePrevious);
    eStatePrevious := eState;
END_IF

METHOD PROTECTED M_Aborted : BOOL // Return
VAR_INPUT
END_VAR
M_Aborted:= FALSE;
END_METHOD

METHOD PROTECTED M_Aborting : BOOL // Return
VAR_INPUT
END_VAR
M_Aborting:= TRUE;
END_METHOD

METHOD PROTECTED M_Completed : BOOL // Return
VAR_INPUT
END_VAR
M_Completed:= TRUE;
END_METHOD

METHOD PROTECTED M_Completing : BOOL // Return
VAR_INPUT
END_VAR
M_Completing:= TRUE;
END_METHOD

METHOD PROTECTED M_Execute : BOOL // Return
VAR_INPUT
END_VAR
M_Execute:= FALSE;
END_METHOD

METHOD PROTECTED M_Held : BOOL // Return
VAR_INPUT
END_VAR
M_Held:= FALSE;
END_METHOD

METHOD PROTECTED M_Holding : BOOL // Return
VAR_INPUT
END_VAR
M_Holding:= TRUE;
END_METHOD

METHOD PROTECTED M_Idle : BOOL // Return
VAR_INPUT
END_VAR
M_Idle:= FALSE;
END_METHOD

METHOD PROTECTED M_Paused : BOOL // Return
VAR_INPUT
END_VAR
M_Paused:= FALSE;
END_METHOD

METHOD PROTECTED M_Pausing : BOOL // Return
VAR_INPUT
END_VAR
M_Pausing:= TRUE;
END_METHOD

METHOD PROTECTED M_Resetting : BOOL // Return
VAR_INPUT
END_VAR
M_Resetting:= TRUE;
END_METHOD

METHOD PROTECTED M_Resuming : BOOL // Return
VAR_INPUT
END_VAR
M_Resuming:= TRUE;
END_METHOD

METHOD PROTECTED M_Starting : BOOL // Return
VAR_INPUT
END_VAR
M_Starting:= TRUE;
END_METHOD

METHOD PROTECTED M_Stopped : BOOL // Return
VAR_INPUT
END_VAR
M_Stopped:= FALSE;
END_METHOD

METHOD PROTECTED M_Stopping : BOOL // Return state complete
VAR_INPUT
END_VAR
M_Stopping:= TRUE;
END_METHOD

METHOD PROTECTED M_Unholding : BOOL // Return
VAR_INPUT
END_VAR
M_Unholding:= TRUE;
END_METHOD

METHOD Protected M_OnState
VAR_INPUT
	eState:							E_State;						// Current state
	eStatePrevious:					E_State;						// Previous state	
END_VAR
// State changed event
fbSequence.M_Reset();
END_METHOD

{attribute 'TcRpcEnable':='1'}
METHOD PUBLIC M_Request : BOOL
VAR_INPUT
	eRequest:	E_Request;
END_VAR
// Request element states
eStateRequest:= eRequest;
M_Request:= True;
END_METHOD

PROPERTY PUBLIC P_Event : I_Event
GET
P_Event:= fbEvent;
END_GET
END_PROPERTY

PROPERTY PUBLIC P_Reflection : I_Reflection
GET
P_Reflection:= fbReflection;
END_GET
END_PROPERTY

PROPERTY PUBLIC P_Sequence : I_Sequence
GET
P_Sequence:= fbSequence;
END_GET
END_PROPERTY

PROPERTY PUBLIC P_State : E_State
GET
P_State:= eState;
END_GET
END_PROPERTY

END_FUNCTION_BLOCK

// Level/FB_Level
FUNCTION_BLOCK FB_Level EXTENDS FB_Element
VAR_INPUT
	fbList:				FB_ListElement;
END_VAR
VAR_OUTPUT
END_VAR
VAR
END_VAR

SUPER^();

METHOD PROTECTED M_Aborting : BOOL (* Return*)
VAR
	nIndex: 	UINT;
END_VAR
M_Aborting:= TRUE;
WHILE nIndex < fbList.nLength DO
    IF fbList.M_Index(nIndex).M_Request(E_Request.Abort) THEN
		;
	ELSE
		M_Aborting:= FALSE;
	END_IF
	nIndex := nIndex + 1;
END_WHILE
END_METHOD

METHOD PUBLIC M_Attach : BOOL
VAR_INPUT
	iComponent:		I_Element;
END_VAR
fbList.M_Add(iComponent);
iComponent.P_Event.P_Logger:= fbEvent.P_Logger;
iComponent.P_Event.P_Observer.M_Attach(THIS^);
fbEvent.fbObserver.M_Attach(iComponent);
M_Attach:= TRUE;
END_METHOD

METHOD PROTECTED M_Completing : BOOL (* Return*)
VAR
	nIndex: 	UINT;
END_VAR
M_Completing:= TRUE;
WHILE nIndex < fbList.nLength DO
    IF fbList.M_Index(nIndex).M_Request(E_Request.Complete) THEN
		;
	ELSE
		M_Completing:= FALSE;
	END_IF
	nIndex := nIndex + 1;
END_WHILE
END_METHOD

METHOD PUBLIC M_Detach : BOOL
VAR_INPUT
END_VAR
END_METHOD

METHOD PROTECTED M_Holding : BOOL (* Return*)
VAR
	nIndex: 	UINT;
END_VAR
M_Holding:= TRUE;
WHILE nIndex < fbList.nLength DO
    IF fbList.M_Index(nIndex).M_Request(E_Request.Hold) THEN
		;
	ELSE
		M_Holding:= FALSE;
	END_IF
	nIndex := nIndex + 1;
END_WHILE
END_METHOD

METHOD PROTECTED M_Pausing : BOOL (* Return*)
VAR
	nIndex: 	UINT;
END_VAR
M_Pausing:= TRUE;
WHILE nIndex < fbList.nLength DO
    IF fbList.M_Index(nIndex).M_Request(E_Request.Pause) THEN
		;
	ELSE
		M_Pausing:= FALSE;
	END_IF
	nIndex := nIndex + 1;
END_WHILE
END_METHOD

METHOD PROTECTED M_Resetting : BOOL (* Return*)
VAR
	nIndex: 	UINT;
END_VAR
M_Resetting:= TRUE;
WHILE nIndex < fbList.nLength DO
    IF fbList.M_Index(nIndex).M_Request(E_Request.Reset) THEN
		;
	ELSE
		M_Resetting:= FALSE;
	END_IF
	nIndex := nIndex + 1;
END_WHILE
END_METHOD

METHOD PROTECTED M_Resuming : BOOL (* Return*)
VAR
	nIndex: 	UINT;
END_VAR
M_Resuming:= TRUE;
WHILE nIndex < fbList.nLength DO
    IF fbList.M_Index(nIndex).M_Request(E_Request.Pause) THEN
		;
	ELSE
		M_Resuming:= FALSE;
	END_IF
	nIndex := nIndex + 1;
END_WHILE
END_METHOD

METHOD PROTECTED M_Starting : BOOL (* Return*)
VAR
	nIndex: 	UINT;
END_VAR
M_Starting:= TRUE;
WHILE nIndex < fbList.nLength DO
    IF fbList.M_Index(nIndex).M_Request(E_Request.Start) THEN
		;
	ELSE
		M_Starting:= FALSE;
	END_IF
	nIndex := nIndex + 1;
END_WHILE
END_METHOD

METHOD PROTECTED M_Stopping : BOOL (* Return state complete*)
VAR
	nIndex: 	UINT;
END_VAR
M_Stopping:= TRUE;
WHILE nIndex < fbList.nLength DO
    IF fbList.M_Index(nIndex).M_Request(E_Request.Reset) THEN
		;
	ELSE
		M_Stopping:= FALSE;
	END_IF
	nIndex := nIndex + 1;
END_WHILE
END_METHOD

METHOD PROTECTED M_Unholding : BOOL (* Return*)
VAR
	nIndex: 	UINT;
END_VAR
M_Unholding:= TRUE;
WHILE nIndex < fbList.nLength DO
    IF fbList.M_Index(nIndex).M_Request(E_Request.Start) THEN
		;
	ELSE
		M_Unholding:= FALSE;
	END_IF
	nIndex := nIndex + 1;
END_WHILE
END_METHOD

PROPERTY PUBLIC P_List : I_ListElement
GET
P_List:= fbList;
END_GET
END_PROPERTY

END_FUNCTION_BLOCK

// List/FB_ListElement
{attribute 'no_explicit_call' := 'do not call this POU directly'} 
FUNCTION_BLOCK FB_ListElement IMPLEMENTS I_ListElement
VAR
	pList: 			POINTER TO I_Element;
	{IF (defined (release))}
    	{attribute 'hide'}
	{END_IF}
	aList:			POINTER TO POINTER TO ARRAY [0..24] OF I_Element:=ADR(pList);
END_VAR
VAR_OUTPUT
	{IF (defined (release))}
    	{attribute 'hide'}
	{END_IF}
	nLength:		INT;	
END_VAR

// https://peterzerlauth.com/

METHOD FB_exit : BOOL
VAR_INPUT
	bInCopyCode : BOOL; // if TRUE, the exit method is called for exiting an instance that is copied afterwards (online change).
END_VAR
M_Clear();
END_METHOD

METHOD PUBLIC M_Add : BOOL
VAR_INPUT
	iObject: 	I_Element;
END_VAR
VAR
	pOldList: 	POINTER TO I_Element;
END_VAR
IF iObject <> 0 THEN
	// First Item
	IF pList = 0 THEN
		nLength:= nLength + 1;
		pList:= __NEW(POINTER TO I_Element,DINT_TO_UDINT(nLength));
	ELSE
		// Item already in List
		IF M_Find(iObject) = -1 THEN
			// backup 
			pOldList:= pList;
			// new Length
			nLength:= nLength + 1;
			// new pointer
			pList:= __NEW(POINTER TO I_Element,DINT_TO_UDINT(nLength));
			// restore
			Memcpy(pList,pOldList, SIZEOF(POINTER TO I_Element)*DINT_TO_UDINT(nLength -1));
			// delete old
			__DELETE(pOldList);
		ELSE
			M_Add:= FALSE;	
			RETURN;
		END_IF
	END_IF
	IF pList = 0 THEN
		RETURN;
	END_IF
	// add new Object
	pList[nLength-1]:= iObject;
	M_Add:= TRUE;
ELSE
	M_Add:= FALSE;	
END_IF
END_METHOD

METHOD PUBLIC M_Clear : BOOL
// Clear
IF pList <> 0 THEN
	nLength:= 0;
	__DELETE(pList);
END_IF
M_Clear:= TRUE;
END_METHOD

METHOD PUBLIC M_Find : DINT
VAR_INPUT
	iObject: 	I_Element;
END_VAR
VAR
	nIndex: 	UINT;
END_VAR
// Find
M_Find := -1;
WHILE nIndex < nLength DO
    IF (pList[nIndex] = iObject) THEN
        M_Find := nIndex;
        RETURN;
    END_IF
	nIndex := nIndex + 1;
END_WHILE
END_METHOD

METHOD PUBLIC M_Index : I_Element
VAR_INPUT
	Index: 	DINT;
END_VAR
VAR
	pTest: 			I_Element:= pList[Index];
END_VAR
// Index
IF Index <= nLength THEN
	M_Index:= pList[Index];
END_IF
END_METHOD

METHOD PUBLIC M_Remove : BOOL
VAR_INPUT
	iObject: 	I_Element;
END_VAR
VAR
	pOldList:			POINTER TO I_Element;
	nPosition: 			DINT;
END_VAR
// Remove
IF iObject <> 0 THEN
	// First Item
	IF nLength >= 0 THEN
		// Item already in List
		nPosition:= M_Find(iObject);
		IF nPosition <> -1 THEN
			// backup 
			pOldList:= pList;
			// new Length
			nLength:= nLength -1;
			// new pointer
			pList:= __NEW(POINTER TO I_Element,DINT_TO_UDINT(nLength));
			// restore lower part
			Memcpy(pList,pOldList, SIZEOF(POINTER TO I_Object) * DINT_TO_UDINT(nPosition));
			//pList[nPosition]:= iObject;
			Memcpy(pList + (SIZEOF(POINTER TO I_Element)*nPosition),pOldList + (SIZEOF(POINTER TO I_Element)*(nPosition + 1)), SIZEOF(POINTER TO I_Element) * DINT_TO_UDINT(nLength - nPosition));
			// delete old
			__DELETE(pOldList);
		ELSE
			M_Remove:= FALSE;	
			RETURN;
		END_IF
	ELSE
		M_Remove:= FALSE;	
		RETURN;
	END_IF
	M_Remove:= TRUE;
ELSE
	M_Remove:= FALSE;	
END_IF
END_METHOD

{attribute 'OPC.UA.DA.Property' := '1'}
{attribute 'monitoring' := 'call'}
PROPERTY PUBLIC P_Length : DINT
GET
P_Length:= nLength;
END_GET
END_PROPERTY

END_FUNCTION_BLOCK

// List/I_ListElement
INTERFACE I_ListElement Extends I_ListBase

METHOD PUBLIC M_Add : BOOL
VAR_INPUT
	iObject: 	I_Element;
END_VAR
END_METHOD

METHOD PUBLIC M_Find : DINT
VAR_INPUT
	iObject: 	I_Element;
END_VAR
END_METHOD

METHOD PUBLIC M_Index : I_Element
VAR_INPUT
	Index: 	DINT;
END_VAR
END_METHOD

METHOD PUBLIC M_Remove : BOOL
VAR_INPUT
	iObject: 	I_Element;
END_VAR
END_METHOD

END_INTERFACE

// List/FB_ListObject
{attribute 'no_explicit_call' := 'do not call this POU directly'} 
FUNCTION_BLOCK FB_ListObject IMPLEMENTS I_ListObject
VAR
	pList: 			POINTER TO I_Object;
	{IF (defined (release))}
    	{attribute 'hide'}
	{END_IF}
	aList:			POINTER TO POINTER TO ARRAY [0..24] OF I_Object:=ADR(pList);
END_VAR
VAR_OUTPUT
	{IF (defined (release))}
    	{attribute 'hide'}
	{END_IF}
	nLength:		INT;	
END_VAR

// https://peterzerlauth.com/

METHOD FB_exit : BOOL
VAR_INPUT
	bInCopyCode : BOOL; // if TRUE, the exit method is called for exiting an instance that is copied afterwards (online change).
END_VAR
M_Clear();
END_METHOD

METHOD PUBLIC M_Add : BOOL
VAR_INPUT
	Object: 	I_Object;
END_VAR
VAR
	pOldList: 	POINTER TO I_Object;
END_VAR
IF Object <> 0 THEN
	// First Item
	IF pList = 0 THEN
		nLength:= nLength + 1;
		pList:= __NEW(POINTER TO I_Object,DINT_TO_UDINT(nLength));
	ELSE
		// Item already in List
		IF M_Find(Object) = -1 THEN
			// backup 
			pOldList:= pList;
			// new Length
			nLength:= nLength + 1;
			// new pointer
			pList:= __NEW(POINTER TO I_Object,DINT_TO_UDINT(nLength));
			// restore
			Memcpy(pList,pOldList, SIZEOF(POINTER TO I_Object)*DINT_TO_UDINT(nLength -1));
			// delete old
			__DELETE(pOldList);
		ELSE
			M_Add:= FALSE;	
			RETURN;
		END_IF
	END_IF
	IF pList = 0 THEN
		RETURN;
	END_IF
	// add new Object
	pList[nLength-1]:= Object;
	M_Add:= TRUE;
ELSE
	M_Add:= FALSE;	
END_IF
END_METHOD

METHOD PUBLIC M_Clear : bool
IF pList <> 0 THEN
	nLength:= 0;
	__DELETE(pList);
END_IF
M_Clear:= TRUE;
END_METHOD

METHOD PUBLIC M_Find : DINT
VAR_INPUT
	Object: 	I_Object;
END_VAR
VAR
	nIndex: 	UINT;
END_VAR
// Object already in List
M_Find := -1;
WHILE nIndex < nLength DO
    IF (pList[nIndex] = Object) THEN
        M_Find := nIndex;
        RETURN;
    END_IF
	nIndex := nIndex + 1;
END_WHILE
END_METHOD

METHOD PUBLIC M_Index : I_Object
VAR_INPUT
	Index: 	DINT;
END_VAR
IF Index <= nLength THEN
	M_Index:= pList[Index];
END_IF
END_METHOD

METHOD PUBLIC M_Remove : BOOL
VAR_INPUT
	Object: 	I_Object;
END_VAR
VAR
	pOldList:			POINTER TO I_Object;
	nPosition: 			DINT;
END_VAR
IF Object <> 0 THEN
	// First Item
	IF nLength >= 0 THEN
		// Item already in List
		nPosition:= M_Find(Object);
		IF nPosition <> -1 THEN
			// backup 
			pOldList:= pList;
			// new Length
			nLength:= nLength -1;
			// new pointer
			pList:= __NEW(POINTER TO I_Object,DINT_TO_UDINT(nLength));
			// restore lower part
			Memcpy(pList,pOldList, SIZEOF(POINTER TO I_Object) * DINT_TO_UDINT(nPosition));
			//pList[nPosition]:= iObject;
			Memcpy(pList + (SIZEOF(POINTER TO I_Object)*nPosition),pOldList + (SIZEOF(POINTER TO I_Object)*(nPosition + 1)), SIZEOF(POINTER TO I_Object) * DINT_TO_UDINT(nLength - nPosition));
			// delete old
			__DELETE(pOldList);
		ELSE
			M_Remove:= FALSE;	
			RETURN;
		END_IF
	ELSE
		M_Remove:= FALSE;	
		RETURN;
	END_IF
	M_Remove:= TRUE;
ELSE
	M_Remove:= FALSE;	
END_IF
END_METHOD

{attribute 'OPC.UA.DA.Property' := '1'}
{attribute 'monitoring' := 'call'}
PROPERTY PUBLIC P_Length : DINT
GET
P_Length:= nLength;
END_GET
END_PROPERTY

END_FUNCTION_BLOCK

// List/I_ListObject
INTERFACE I_ListObject Extends I_ListBase

METHOD PUBLIC M_Add : BOOL
VAR_INPUT
	Object: 	I_Object;
END_VAR
END_METHOD

METHOD PUBLIC M_Find : DINT
VAR_INPUT
	Object: 	I_Object;
END_VAR
END_METHOD

METHOD PUBLIC M_Index : I_Object
VAR_INPUT
	Index: 	DINT;
END_VAR
END_METHOD

METHOD PUBLIC M_Remove : BOOL
VAR_INPUT
	Object: 	I_Object;
END_VAR
END_METHOD

END_INTERFACE

// Logger/FB_FileLogger
FUNCTION_BLOCK FB_FileLogger VAR_GENERIC CONSTANT nMaxLength: UINT := 10; END_VAR IMPLEMENTS I_Logger
VAR_INPUT
	sPathName:					STRING;
END_VAR
VAR
	nLength:					DINT;
	aEvent:						ARRAY [0..nMaxLength - 1] OF ST_Event;
	fbFile:						FB_File;
	bWriteLine: BOOL;
END_VAR

// https://peterzerlauth.com/

fbFile();

IF fbFile.P_Open THEN
	;
ELSE
	fbFile.M_Create(sPathName);
END_IF

IF bWriteLine THEN
	bWriteLine:= NOT fbFile.M_AppendLine('Test');
END_IF

METHOD PUBLIC M_Delete : BOOL
VAR_INPUT
	nIndex: 			DINT;
END_VAR
// new Length
nLength:= nLength -1;
//pList[nPosition]:= iObject;
Memcpy(ADR(aEvent[nIndex]), ADR(aEvent[nIndex +1]), SIZEOF(POINTER TO ST_Event) * DINT_TO_UDINT(nMaxLength - nIndex));
END_METHOD

METHOD PUBLIC M_Find : DINT
VAR_INPUT
	stEvent:	ST_Event;
END_VAR
VAR 
	nIndex:		DINT;
END_VAR
// Find event in buffer
M_Find := -1;
WHILE nIndex < nLength DO
	IF (aEvent[nIndex].iSource = stEvent.iSource) AND_THEN
    	(aEvent[nIndex].eEventType = stEvent.eEventType) AND_THEN
		(aEvent[nIndex].sInstance = stEvent.sInstance) AND_THEN
		(aEvent[nIndex].sMessage = stEvent.sMessage) THEN
        M_Find := nIndex;
        RETURN;
    END_IF
	nIndex := nIndex + 1;
END_WHILE
END_METHOD

METHOD PUBLIC M_Log
VAR_INPUT
	stEvent:		ST_Event;
END_VAR
VAR
	nIndex:			DINT;
END_VAR
IF (nIndex:=  M_Find(stEvent)) >= 0 THEN
	// Update existing events
	aEvent[nIndex].sArguments:= stEvent.sArguments;
	aEvent[nIndex].sDefault:= stEvent.sDefault;
	aEvent[nIndex].sClass:= stEvent.sClass;
	aEvent[nIndex].stFlags:= stEvent.stFlags;
	
ELSE
	// add new event
	aEvent[nLength]:= stEvent;
	nLength:= nLength + 1;
	
// 	fbFile.M_AppendLine(stEvent.eEventType
END_IF
END_METHOD

METHOD PUBLIC M_Reset
VAR_INPUT
END_VAR
// Reset all events
nLength:= 0;
Memset(ADR(aEvent), 0, SIZEOF(aEvent));
END_METHOD

END_FUNCTION_BLOCK

// Utils/File/FB_File
{attribute 'no_explicit_call'} 
FUNCTION_BLOCK FB_File
VAR
    fbCreateDir:	FB_CreateDir;
	fbOpen:			FB_FileOpen;
	fbRead:			FB_FileRead;
	fbLoad:			FB_FileLoad;
	fbWrite:		FB_FileWrite;
	fbClose:		FB_FileClose;
	fbDelete:		FB_FileDelete;
END_VAR
VAR_OUTPUT
	nError:			UDINT;
END_VAR

// https://peterzerlauth.com/
fbCreateDir();
fbLoad();
fbOpen();
fbClose();
fbDelete();
fbWrite();
fbRead();

METHOD PUBLIC M_Append : BOOL
VAR_INPUT
	Text:			STRING(255);
END_VAR
IF fbWrite.bExecute THEN
	IF fbWrite.bError THEN
		nError:= fbWrite.nErrId;
		fbWrite.bExecute:= FALSE;
	ELSIF fbWrite.bBusy THEN
		;
	ELSE
		M_Append:= TRUE;
		fbWrite.bExecute:= FALSE;
	END_IF
ELSE
	fbWrite.bExecute:= TRUE;
	fbWrite.pWriteBuff:= ADR(Text);
	fbWrite.cbWriteLen:= INT_TO_UDINT(Len(Text));
END_IF
END_METHOD

METHOD PUBLIC M_AppendLine : BOOL
VAR_INPUT
	Text:			STRING(255);
END_VAR
Text:= Concat(Text, '$R');
M_AppendLine:= M_Append(Text);
END_METHOD

METHOD PUBLIC M_Close : BOOL
VAR_INPUT
END_VAR
IF fbClose.bExecute THEN
	IF fbClose.hFile = 0 THEN
		fbClose.bExecute:= FALSE;
		M_Close:= TRUE;
	ELSIF fbClose.bError THEN
		fbClose.bExecute:= FALSE;
		nError:= fbClose.nErrId;
	ELSIF fbClose.bBusy THEN
		;
	ELSE
		nError:= 0;	
		fbRead.hFile:= 0;
		fbWrite.hFile:= 0;
		fbClose.hFile:= 0;
		fbClose.bExecute:= FALSE;
		M_Close:= TRUE;
	END_IF
ELSE
	fbClose.bExecute:= TRUE;
END_IF
END_METHOD

METHOD PUBLIC M_Create : BOOL
VAR_INPUT
	PathName:		STRING(255);
END_VAR
VAR
	nTemp: INT;
END_VAR
VAR_INST
	nPosition: INT;
END_VAR
nTemp := FIND(RIGHT(PathName, LEN(PathName) - nPosition), '\');
if nTemp <> 0 then
	IF fbCreateDir.bExecute THEN
		IF NOT fbCreateDir.bBusy THEN
			nPosition := nPosition + nTemp;
			fbCreateDir.bExecute:= FALSE;
		END_IF
	ELSE
		fbCreateDir.bExecute:= TRUE;
		fbCreateDir.ePath:= PATH_GENERIC;
		fbCreateDir.sPathName:= Left(PathName, nPosition + nTemp);
	END_IF
ELSE
	IF M_Open(PathName) THEN
		M_Create:= TRUE;
		nPosition:= 0;
	END_IF
END_IF
END_METHOD

METHOD PUBLIC M_Delete : BOOL
VAR_INPUT
	PathName:		STRING(255);
END_VAR
IF fbDelete.bExecute THEN
	IF fbDelete.bError THEN
		fbDelete.bExecute:= FALSE;
		M_Delete:= TRUE;
	ELSIF fbDelete.bBusy THEN
		;
	ELSE
		fbDelete.bExecute:= FALSE;
		M_Delete:= TRUE;
	END_IF
ELSE
	fbDelete.bExecute:= TRUE;
	fbDelete.sPathName:= PathName;
	fbDelete.ePath:= E_OpenPath.PATH_GENERIC;
END_IF
END_METHOD

METHOD PUBLIC M_Load : BOOL
VAR_INPUT
	PathName:		STRING(255);
	Value:			ANY;
END_VAR
IF fbLoad.bExecute THEN
	IF fbLoad.bError THEN
		nError:= fbLoad.nErrId;
		fbLoad.bExecute:= FALSE;
	ELSIF fbLoad.bBusy THEN
		;
	ELSE
		M_Load:= TRUE;
	END_IF
ELSE
	fbLoad.sPathName:= PathName;
	fbLoad.bExecute:= TRUE;
	fbLoad.pReadBuff:= Value.pValue;
	fbLoad.cbReadLen:= DINT_TO_UDINT(Value.diSize);
END_IF
END_METHOD

METHOD PUBLIC M_Open : BOOL
VAR_INPUT
	PathName:		STRING(255);
END_VAR
// Check if the file open should be executed
IF fbOpen.bExecute THEN
    // Check the file opening process
    IF fbOpen.bError THEN
        // Store the error ID and stop the execution
        nError:= fbOpen.nErrId;
        fbOpen.bExecute:= FALSE;
        
    // If the process is still busy, do nothing and wait
    ELSIF fbOpen.bBusy THEN
        ;
        
    // If the file has been successfully opened
    ELSIF fbOpen.hFile <> 0 THEN    
        // Assign the file handle
        fbRead.hFile:= fbOpen.hFile;
        fbWrite.hFile:= fbOpen.hFile;
        fbClose.hFile:= fbOpen.hFile;
        fbOpen.bExecute:= FALSE;
        // File is open
        M_Open:= TRUE;
    END_IF    
ELSE
    // If the file handle is invalid (e.g., the file is not open)
    IF fbOpen.hFile = 0 THEN
        // file is open
        M_Open:= TRUE;    
    ELSE
        // Start the file opening process with the specified path and mode
        fbOpen.bExecute:= TRUE;
        fbOpen.sPathName:= PathName;
        fbOpen.nMode:= (FOPEN_MODEAPPEND OR FOPEN_MODEPLUS OR FOPEN_MODETEXT);    
    END_IF
END_IF
END_METHOD

METHOD PUBLIC M_Read : BOOL
VAR_INPUT
	Value:		ANY;
END_VAR
IF fbRead.bExecute THEN
	IF fbRead.bError THEN
		nError:= fbRead.nErrId;
		fbRead.bExecute:= FALSE;
	ELSIF fbRead.bBusy THEN
		;
	ELSE
		fbRead.bExecute:= FALSE;
		M_Read:= TRUE;
	END_IF
ELSE
	fbRead.bExecute:= TRUE;
	fbRead.pReadBuff:= Value.pValue;
	fbRead.cbReadLen:= DINT_TO_UDINT(Value.diSize);
END_IF
END_METHOD

METHOD PUBLIC M_Write : BOOL
VAR_INPUT
	Value:		ANY;
END_VAR
IF fbWrite.bExecute THEN
	IF fbWrite.bError THEN
		nError:= fbWrite.nErrId;
		fbWrite.bExecute:= FALSE;
	ELSIF fbWrite.bBusy THEN
		M_Write:= FALSE;
	ELSE
		M_Write:= TRUE;
		fbWrite.bExecute:= FALSE;
	END_IF
ELSE
	fbWrite.bExecute:= TRUE;
	MEMCPY(ADR(fbWrite.cbWrite), Value.pValue, SIZEOF(POINTER TO BYTE));
	fbWrite.cbWriteLen:= DINT_TO_UDINT(Value.diSize);
END_IF
END_METHOD

PROPERTY PUBLIC P_Error : UDINT
GET
P_Error:= nError;
END_GET
END_PROPERTY

PROPERTY PUBLIC P_Open : Bool
GET
P_Open:= fbOpen.hFile <> 0;
END_GET
END_PROPERTY

END_FUNCTION_BLOCK

// Logger/FB_Logger
FUNCTION_BLOCK FB_Logger VAR_GENERIC CONSTANT nMaxLength: UINT := 10; END_VAR IMPLEMENTS I_Logger
VAR
	nLength:					DINT;
	aEvent:						ARRAY [0..nMaxLength - 1] OF ST_Event;
	nIndex: 					DINT;
	nTimestamp: 				ULINT;
END_VAR

// https://peterzerlauth.com/
// Execute each secound
IF nTimestamp <= F_GetSystemTime() THEN
	nTimestamp:= F_GetSystemTime() + 10000000;
	nIndex:= 0;
	WHILE nIndex < nLength DO
		IF aEvent[nIndex].stFlags.bActive THEN
			IF aEvent[nIndex].stFlags.bRemove THEN
				aEvent[nIndex].stFlags.bActive:= FALSE;
			END_IF
		ELSE
			M_Delete(nIndex);
		END_IF
		nIndex := nIndex + 1;
	END_WHILE
END_IF

METHOD PUBLIC M_Delete : BOOL
VAR_INPUT
	nIndex: 			DINT;
END_VAR
// new Length
nLength:= nLength -1;
//pList[nPosition]:= iObject;
Memcpy(ADR(aEvent[nIndex]), ADR(aEvent[nIndex +1]), SIZEOF(POINTER TO ST_Event) * DINT_TO_UDINT(nMaxLength - nIndex));
END_METHOD

METHOD PUBLIC M_Find : DINT
VAR_INPUT
	stEvent:	ST_Event;
END_VAR
VAR 
	nIndex:		DINT;
END_VAR
// Find event in buffer
M_Find := -1;
WHILE nIndex < nLength DO
	IF (aEvent[nIndex].iSource = stEvent.iSource) AND_THEN
    	(aEvent[nIndex].eEventType = stEvent.eEventType) AND_THEN
		(aEvent[nIndex].sInstance = stEvent.sInstance) AND_THEN
		(aEvent[nIndex].sMessage = stEvent.sMessage) THEN
        M_Find := nIndex;
        RETURN;
    END_IF
	nIndex := nIndex + 1;
END_WHILE
END_METHOD

METHOD PUBLIC M_Log
VAR_INPUT
	stEvent:		ST_Event;
END_VAR
VAR
	nIndex:			DINT;
END_VAR
IF (nIndex:=  M_Find(stEvent)) >= 0 THEN
	// Update existing events
	aEvent[nIndex].sArguments:= stEvent.sArguments;
	aEvent[nIndex].sDefault:= stEvent.sDefault;
	aEvent[nIndex].sClass:= stEvent.sClass;
	aEvent[nIndex].stFlags:= stEvent.stFlags;
ELSE
	// add new event
	aEvent[nLength]:= stEvent;
	nLength:= nLength + 1;
END_IF
END_METHOD

METHOD PUBLIC M_Reset
VAR_INPUT
END_VAR
// Reset all events
nLength:= 0;
Memset(ADR(aEvent), 0, SIZEOF(aEvent));
END_METHOD

END_FUNCTION_BLOCK

// Logger/FB_LoggingProvider
{attribute 'no_explicit_call' := 'do not call this POU directly'} 
FUNCTION_BLOCK FB_LoggingProvider IMPLEMENTS I_Logger
VAR
	{IF (defined (release))}
    	{attribute 'hide'}
	{END_IF}
	nLength:		INT;
	pList: 			POINTER TO I_Logger;
	{IF (defined (release))}
    	{attribute 'hide'}
	{END_IF}
	aList:			POINTER TO POINTER TO ARRAY [0..24] OF I_Logger:=ADR(pList);
END_VAR

// https://peterzerlauth.com/

METHOD FB_exit : BOOL
VAR_INPUT
	bInCopyCode : BOOL; // if TRUE, the exit method is called for exiting an instance that is copied afterwards (online change).
END_VAR
M_Clear();
END_METHOD

METHOD PUBLIC M_Add : BOOL
VAR_INPUT
	Logger: 	I_Logger;
END_VAR
VAR
	pOldList: 	POINTER TO I_Logger;
END_VAR
IF Logger <> 0 THEN
	// First Item
	IF pList = 0 THEN
		nLength:= nLength + 1;
		pList:= __NEW(POINTER TO I_Logger,DINT_TO_UDINT(nLength));
	ELSE
		// Item already in List
		IF M_Find(Logger) = -1 THEN
			// backup 
			pOldList:= pList;
			// new Length
			nLength:= nLength + 1;
			// new pointer
			pList:= __NEW(POINTER TO I_Logger,DINT_TO_UDINT(nLength));
			// restore
			Memcpy(pList,pOldList, SIZEOF(POINTER TO I_Logger)*DINT_TO_UDINT(nLength -1));
			// delete old
			__DELETE(pOldList);
		ELSE
			M_Add:= FALSE;	
			RETURN;
		END_IF
	END_IF
	IF pList = 0 THEN
		RETURN;
	END_IF
	// add new Object
	pList[nLength-1]:= Logger;
	M_Add:= TRUE;
ELSE
	M_Add:= FALSE;	
END_IF
END_METHOD

METHOD PUBLIC M_Clear : bool
IF pList <> 0 THEN
	nLength:= 0;
	__DELETE(pList);
END_IF
M_Clear:= TRUE;
END_METHOD

METHOD PUBLIC M_Find : DINT
VAR_INPUT
	Logger: 	I_Logger;
END_VAR
VAR
	nIndex: 	UINT;
END_VAR
// Object already in List
M_Find := -1;
WHILE nIndex < nLength DO
    IF (pList[nIndex] = Logger) THEN
        M_Find := nIndex;
        RETURN;
    END_IF
	nIndex := nIndex + 1;
END_WHILE
END_METHOD

METHOD PUBLIC M_Index : I_Logger
VAR_INPUT
	Index: 	DINT;
END_VAR
IF Index <= nLength THEN
	M_Index:= pList[Index];
END_IF
END_METHOD

METHOD public M_Log
VAR_INPUT
	stEvent	: ST_Event;
END_VAR
VAR
	nIndex:		INT;
END_VAR
WHILE nIndex < nLength DO
    pList[nIndex].M_Log(stEvent);
	nIndex := nIndex + 1;
END_WHILE
END_METHOD

METHOD PUBLIC M_Remove : BOOL
VAR_INPUT
	Object: 	I_Logger;
END_VAR
VAR
	pOldList:			POINTER TO I_Logger;
	nPosition: 			DINT;
END_VAR
IF Object <> 0 THEN
	// First Item
	IF nLength >= 0 THEN
		// Item already in List
		nPosition:= M_Find(Object);
		IF nPosition <> -1 THEN
			// backup 
			pOldList:= pList;
			// new Length
			nLength:= nLength -1;
			// new pointer
			pList:= __NEW(POINTER TO I_Logger,DINT_TO_UDINT(nLength));
			// restore lower part
			Memcpy(pList,pOldList, SIZEOF(POINTER TO I_Logger) * DINT_TO_UDINT(nPosition));
			//pList[nPosition]:= iObject;
			Memcpy(pList + (SIZEOF(POINTER TO I_Logger)*nPosition),pOldList + (SIZEOF(POINTER TO I_Logger)*(nPosition + 1)), SIZEOF(POINTER TO I_Logger) * DINT_TO_UDINT(nLength - nPosition));
			// delete old
			__DELETE(pOldList);
		ELSE
			M_Remove:= FALSE;	
			RETURN;
		END_IF
	ELSE
		M_Remove:= FALSE;	
		RETURN;
	END_IF
	M_Remove:= TRUE;
ELSE
	M_Remove:= FALSE;	
END_IF
END_METHOD

METHOD public M_Reset
VAR
	nIndex:		INT;
END_VAR
WHILE nIndex < nLength DO
    pList[nIndex].M_Reset();
	nIndex := nIndex + 1;
END_WHILE
END_METHOD

{attribute 'OPC.UA.DA.Property' := '1'}
{attribute 'monitoring' := 'call'}
PROPERTY PUBLIC P_Length : DINT
GET
P_Length:= nLength;
END_GET
END_PROPERTY

END_FUNCTION_BLOCK

// Module/FB_Module
FUNCTION_BLOCK FB_Module EXTENDS FB_Element IMPLEMENTS I_Module
VAR_INPUT
END_VAR
VAR_OUTPUT
END_VAR
VAR
	fbLogging:					FB_LoggingProvider;
	fbLogger:					FB_Logger<20>;
	{attribute 'OPC.UA.DA' := '1'}
	{attribute 'OPC.UA.DA.Access' := '1'}
	eModeRequest:					E_Mode:= E_Mode.Automatic;				// Requested mod
	{attribute 'OPC.UA.DA' := '1'}
	{attribute 'OPC.UA.DA.Access' := '2'}
	eMode:							E_Mode;				// Current mode
	{attribute 'hide'}
	eModePrevious:					E_Mode;				// Previous mode
	
	fbLevel1:					FB_Level;
	fbLevel2:					FB_Level;
	fbLevel3:					FB_Level;
	fbLevel4:					FB_Level;
END_VAR

// https://peterzerlauth.com/
SUPER^();

fbLevel1();
fbLevel2();
fbLevel3();
fbLevel4();

// Detect mode changes
IF eModeRequest <> E_Mode.Undefined THEN
	IF eMode <> eModeRequest THEN
		eModePrevious:= eMode;
		eMode:= eModeRequest;
		M_OnMode(eMode, eModePrevious);
	END_IF
END_IF
eModeRequest:= E_Mode.Undefined;

METHOD PROTECTED M_Aborting : BOOL (* Return*)
M_Aborting:= 	fbLevel4.M_Request(E_Request.Abort) AND
 				fbLevel3.M_Request(E_Request.Abort) AND
				fbLevel2.M_Request(E_Request.Abort) AND
				fbLevel1.M_Request(E_Request.Abort);
END_METHOD

METHOD PROTECTED M_Completing : BOOL (* Return*)
M_Completing:= 	fbLevel2.M_Request(E_Request.Complete) AND
				fbLevel1.M_Request(E_Request.Complete);
END_METHOD

METHOD PROTECTED M_Holding : BOOL (* Return*)
M_Holding:= fbLevel1.M_Request(E_Request.Hold);
END_METHOD

METHOD PROTECTED M_Idle : BOOL (* Return*)
fbLogging.M_Add(fbLogger);

fbLevel4.P_Event.P_Logger:= fbLogging;
fbLevel3.P_Event.P_Logger:= fbLogging;
fbLevel2.P_Event.P_Logger:= fbLogging;
fbLevel1.P_Event.P_Logger:= fbLogging;

fbLevel4.M_Attach(fbLevel3);
fbLevel4.M_Attach(fbLevel2);
fbLevel4.M_Attach(fbLevel1);

fbLevel3.M_Attach(fbLevel2);
fbLevel3.M_Attach(fbLevel1);

fbLevel2.M_Attach(fbLevel1);

fbEvent.fbObserver.M_Attach(fbLevel1);
END_METHOD

{attribute 'TcRpcEnable':='1'}
METHOD PUBLIC M_Mode : BOOL
VAR_INPUT
	eMode:		E_Mode;
END_VAR
IF THIS^.eMode = eMode THEN
	M_Mode:= TRUE;
ELSE
	eModeRequest:= eMode;	
END_IF
END_METHOD

METHOD PROTECTED M_OnMode
VAR_INPUT
	eMode:							E_Mode;						// Current mode
	eModePrevious:					E_Mode;						// Previous mode	
END_VAR
CASE eMode OF
	E_Mode.Semiauto, E_Mode.Automatic:
		IF eModePrevious = E_Mode.Manual THEN
			fbEvent.M_AddSTRING(TO_STRING(eModePrevious));
			fbEvent.M_AddSTRING(TO_STRING(eMode));
			fbEvent.M_Abort('Module mode changed form %s to %s', 1002);
		END_IF
	E_Mode.Manual:
		;
END_CASE
END_METHOD

METHOD PROTECTED M_Resetting : BOOL (* Return*)
M_Resetting:= 	fbLevel4.M_Request(E_Request.Reset) AND
 				fbLevel3.M_Request(E_Request.Reset) AND
				fbLevel2.M_Request(E_Request.Reset) AND
				fbLevel1.M_Request(E_Request.Reset);
END_METHOD

METHOD PROTECTED M_Starting : BOOL
VAR_INPUT
END_VAR
M_Starting:= 	fbLevel4.M_Request(E_Request.Start) AND_THEN
 				fbLevel3.M_Request(E_Request.Start) AND_THEN
				fbLevel2.M_Request(E_Request.Start) AND_THEN
				fbLevel1.M_Request(E_Request.Start);
END_METHOD

METHOD PROTECTED M_Stopping : BOOL (* Return state complete*)
M_Stopping:= 	fbLevel3.M_Request(E_Request.Stop) AND
				fbLevel2.M_Request(E_Request.Stop) AND
				fbLevel1.M_Request(E_Request.Stop);
END_METHOD

METHOD PROTECTED M_Unholding : BOOL (* Return*)
M_Unholding:= fbLevel1.M_Request(E_Request.Start);
END_METHOD

PROPERTY PUBLIC P_Mode : E_Mode
GET
P_Mode:= eMode;
END_GET
END_PROPERTY

END_FUNCTION_BLOCK

// Module/I_Module
INTERFACE I_Module EXTENDS I_Element

METHOD PUBLIC M_Mode : BOOL
VAR_INPUT
	eMode:		E_Mode;
END_VAR
END_METHOD

PROPERTY PUBLIC P_Mode : E_Mode
GET
END_GET
END_PROPERTY

END_INTERFACE

// Object/FB_Object
FUNCTION_BLOCK FB_Object IMPLEMENTS I_Object
VAR_INPUT
END_VAR
VAR_OUTPUT
END_VAR
VAR
END_VAR

END_FUNCTION_BLOCK

// Utils/File/I_File
INTERFACE I_File

METHOD PUBLIC M_Append : BOOL
VAR_INPUT
	sText:			STRING(255);
END_VAR
END_METHOD

METHOD PUBLIC M_AppendLine : BOOL
VAR_INPUT
	sText:			STRING(255);
END_VAR
END_METHOD

METHOD PUBLIC M_Close : BOOL
VAR_INPUT
END_VAR
END_METHOD

METHOD PUBLIC M_Create : BOOL
VAR_INPUT
	sPathName:		T_MaxString;
END_VAR
END_METHOD

METHOD PUBLIC M_Delete : BOOL
VAR_INPUT
	sPathName:		T_MaxString;
END_VAR
END_METHOD

METHOD PUBLIC M_Load : BOOL
VAR_INPUT
	sPathName:		T_MaxString;
	pData:			PVOID;
	nData:			UDINT;
END_VAR
END_METHOD

METHOD PUBLIC M_Open : BOOL
VAR_INPUT
	sPathName:		T_MaxString;
END_VAR
END_METHOD

METHOD PUBLIC M_Read : BOOL
VAR_INPUT
	Value:		ANY;
END_VAR
END_METHOD

METHOD PUBLIC M_Write : BOOL
VAR_INPUT
	Value:		ANY;
END_VAR
END_METHOD

PROPERTY PUBLIC P_Error : UDINT
GET
END_GET
END_PROPERTY

PROPERTY PUBLIC P_Open : Bool
GET
END_GET
END_PROPERTY

END_INTERFACE

// Utils/FB_Debounce
FUNCTION_BLOCK FB_Debounce 
VAR_INPUT
	bInput:				BOOL;
	tTime:				TIME;
END_VAR
VAR_OUTPUT
	bValue:				BOOL;
END_VAR
VAR
	fbTimerOn:			Ton;
	fbTimerOff:			Ton;
END_VAR

// https://peterzerlauth.com/
IF bInput THEN
	fbTimerOn(IN:= TRUE, PT:= tTime);
	fbTimerOff(IN:= FALSE);
	IF fbTimerOn.Q THEN
		bValue:= TRUE;
	END_IF
ELSE
	fbTimerOff(IN:= TRUE, PT:= tTime);
	fbTimerOn(IN:= FALSE);
	IF fbTimerOff.Q THEN
		bValue:= FALSE;
	END_IF	
END_IF

PROPERTY PUBLIC P_Value : BOOL
GET
P_Value:= bValue;
END_GET
END_PROPERTY

END_FUNCTION_BLOCK
